{attribute 'qualified_only'}
VAR_GLOBAL
END_VAR

(* stored: Version 1.1.0.1, ProductVersion 3.1.4024.11
   GVL Hardware_A24: Id {27bc0540-0d18-48f2-9be8-1f3dc031eed7} *)
